PROGRAM DAS_MotionSync
VAR
END_VAR

AxisInterface_Type03();
M_InputMapping();

METHOD M_InputMapping
VAR_INPUT
END_VAR
// TurnTable Axis sensor
arAxisCtrl_gb[AxisNo.TurnTable].SetupMode.bHomeSignal := NOT GVL_Input.uniDI.stDI.bTurnTable_Axis_HomeSensor;
// RoundBelt Axis sensor
arAxisCtrl_gb[AxisNo.RoundBelt].SetupMode.bHomeSignal := GVL_Input.uniDI.stDI.bRoundBelt_Axis_HomeSensor;
// Allocate Robot X Axis
arAxisCtrl_gb[AxisNo.Allocate_X].SetupMode.bPosLimitSignal:= NOT GVL_Input.uniDI.stDI.bAllocateRobot_Xaxis_PosLimit;
arAxisCtrl_gb[AxisNo.Allocate_X].SetupMode.bNegimitSignal:=  NOT GVL_Input.uniDI.stDI.bAllocateRobot_Xaxis_NegLimit;

//arAxisCtrl_gb[AxisNo.Allocate_Y].SetupMode.bHomeSignal:= ;
	//arAxisCtrl_gb[AxisNo.Allo cate_Y].SetupMode.bNegimitSignal:=;

arAxisCtrl_gb[AxisNo.OutRobot_X].SetupMode.bHomeSignal:= GVL_Input.uniDI.stDI.bOutRobot_Xaxis_HomeSensor;
arAxisCtrl_gb[AxisNo.OutRobot_X].SetupMode.bPosLimitSignal:=  NOT GVL_Input.uniDI.stDI.bOutRobot_Xaxis_PosLimit;
arAxisCtrl_gb[AxisNo.OutRobot_X].SetupMode.bNegimitSignal:=  NOT GVL_Input.uniDI.stDI.bOutRobot_Xaxis_NegLimit;

arAxisCtrl_gb[AxisNo.OutRobot_Y].SetupMode.bHomeSignal:= GVL_Input.uniDI.stDI.bOutRobot_Yaxis_HomeSensor;
arAxisCtrl_gb[AxisNo.OutRobot_Y].SetupMode.bPosLimitSignal:=  NOT GVL_Input.uniDI.stDI.bOutRobot_Yaxis_PosLimit;
arAxisCtrl_gb[AxisNo.OutRobot_Y].SetupMode.bNegimitSignal:=  NOT GVL_Input.uniDI.stDI.bOutRobot_Yaxis_NegLimit;

arAxisCtrl_gb[AxisNo.RackMotor].SetupMode.bNegimitSignal := NOT GVL_Input.uniDI.stDI.bStackPush_DCMotor_NegLimit;
arAxisCtrl_gb[AxisNo.RackMotor].SetupMode.bPosLimitSignal := not GVL_Input.uniDI.stDI.bStackPush_DCMotor_PosLimit;
END_METHOD

END_PROGRAM

(* stored: Version 1.1.0.1, ProductVersion 3.1.4024.13
   POU DAS_MotionSync: Id {445b1210-9ce8-43e0-9271-a5543f119091}, SpecialFunc None
   Method M_InputMapping: Id {e123f82b-4486-455a-8ca2-11803ec326de} *)
